Staubli VAL3: listadd.pgx

public program listadd(string& x_sItems[] (dimensions=1))
  local num i
  local num l_nSize
begin
  //---------------------------------
  // insert x_sItems into the list
  //---------------------------------
  //
  // x_sItems:      Items to add
  //
  //---------------------------------
  // Staubli copyright 2005
  //                By toneage
  //[Public]-------------------------
  //
  //
  for i=0 to (size(x_sItems)-1)
    if (size(sItems)!=1 or sItems!="") and x_sItems[i]!=""
      insert(sItems[size(sItems)])
      insert(bReadWrite[size(bReadWrite)])
    endIf
    if x_sItems[i]!=""
      sItems[size(sItems)-1]=x_sItems[i]
      // for default the RW is true
      bReadWrite[size(bReadWrite)-1]=true
    endIf
  endFor
end
